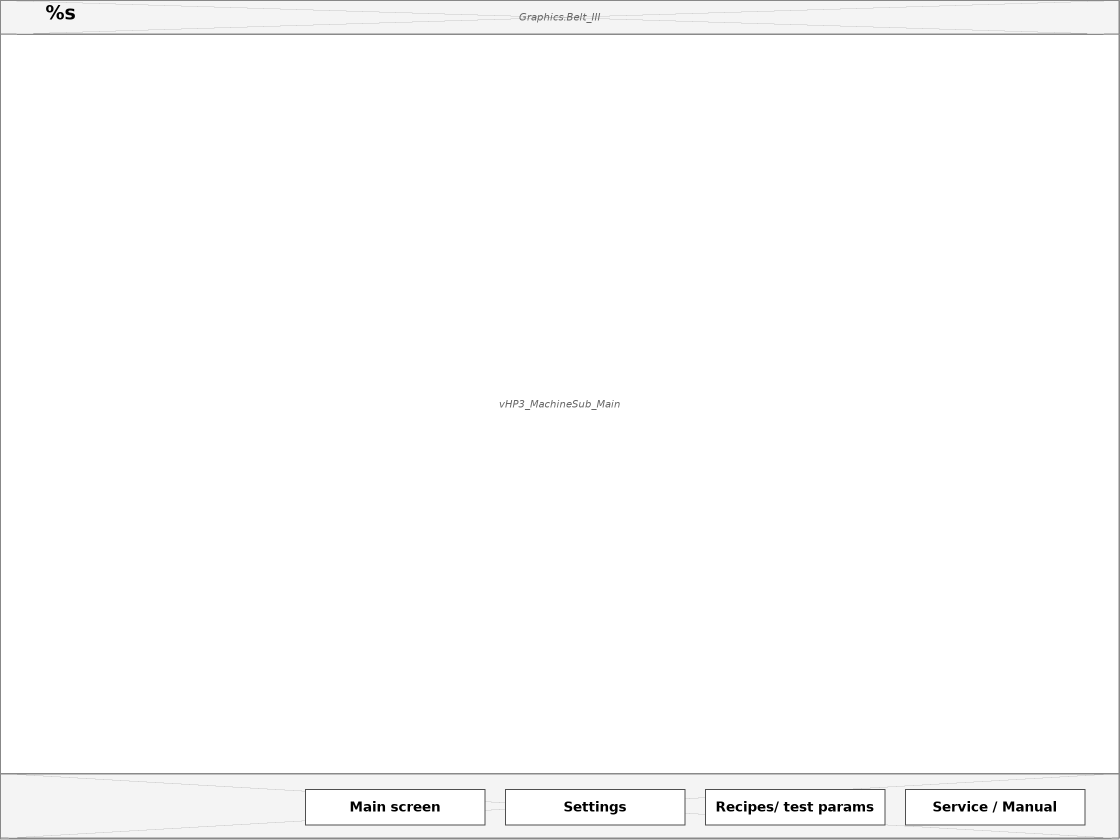
VISUALIZATION vHP3_MainMachine  // 1120x840
VAR_IN_OUT
	fbHP: fbHPv3_Control;
END_VAR
    Image (0,0 1120x34), invisible if: fbHP.iMachineNumber <> 2, image: Graphics.Belt_II
    Image (0,773 1120x65), invisible if: fbHP.iMachineNumber <> 3, image: Graphics.Belt_III
    Image (0,773 1120x65), invisible if: fbHP.iMachineNumber <> 1, image: Graphics.Belt_I
    Image (0,773 1120x65), invisible if: fbHP.iMachineNumber <> 2, image: Graphics.Belt_II
    Image (0,0 1120x34), invisible if: fbHP.iMachineNumber <> 1, image: Graphics.Belt_I
    Rectangle (305,789 180x36), "Main screen"
        OnMouseClick: FrameSelectionChange Selection=SelectedFrame=2d948332-6323-4ce4-b5f8-a8f9ee9afdb0, GlobSel=AssignType=Expression, SelType=Locally
        OnMouseClick: execute { fbHP.iHMI_ActFrame := 0; }
    Rectangle (505,789 180x36), "Settings"
        OnMouseClick: FrameSelectionChange Selection=SelectedFrame=2d948332-6323-4ce4-b5f8-a8f9ee9afdb0, Selection=1, GlobSel=AssignType=Expression, SelType=Locally
        OnMouseClick: execute { fbHP.iHMI_ActFrame := 1; }
    Rectangle (905,789 180x36), "Service / Manual"
        OnMouseClick: FrameSelectionChange Selection=SelectedFrame=2d948332-6323-4ce4-b5f8-a8f9ee9afdb0, Selection=3, GlobSel=AssignType=Expression, SelType=Locally
        OnMouseClick: execute { fbHP.iHMI_ActFrame := 3; }
    Rectangle (705,789 180x36), "Recipes/ test params"
        OnMouseClick: FrameSelectionChange Selection=SelectedFrame=2d948332-6323-4ce4-b5f8-a8f9ee9afdb0, Selection=2, GlobSel=AssignType=Expression, SelType=Locally
        OnMouseClick: execute { fbHP.iHMI_ActFrame := 2; }
    Frame (0,34 1120x740)
        shows vHP3_MachineSub_Main(fbHP := fbHP)
        shows vHP3_MachineSub_Settings(fbHP := fbHP)
        shows vHP3_MachineSub_TestParams(fbHP := fbHP)
        shows vHP3_MachineSub_Service(fbHP := fbHP)
    Image (0,0 1120x34), invisible if: fbHP.iMachineNumber <> 3, image: Graphics.Belt_III
    RoundedRectangle (10,0 716x32), "%s", text list: 'tlHPv3', text index: fbHP.iMachineNumber
END_VISUALIZATION

(* stored: Version 1.1.0.1, ProductVersion 3.1.4024.13
   Visu vHP3_MainMachine: Id {2a335ca7-7433-480e-a6e3-dec8b3e47b85} *)
